FUNCTION_BLOCK FB_Pt100
VAR_INPUT
	Raw : INT;
END_VAR
VAR_OUTPUT
	TempCelsius : REAL;
	TempFaranheit : REAL;
END_VAR

// Card settings: 3-wire, 0,1°C precision, pt100

TempCelsius:= Raw/10;
TempFaranheit := (TempCelsius*9/5)+32;

END_FUNCTION_BLOCK

(* stored: Version 1.1.0.1, ProductVersion 3.1.4024.9
   POU FB_Pt100: Id {9ce2ec01-883c-4d32-95bb-2a3410b18095}, SpecialFunc None *)
